// TIA Portal V20 export
VAR_GLOBAL   // PLC tag table "temp"
END_VAR
